FUNCTION_BLOCK FB_ROB_AMR EXTENDS FB_ROB IMPLEMENTS ITF_2_AMR
VAR_INPUT
END_VAR
VAR_OUTPUT
	visStatus: stVisStatusAMR;
	bTargetreached: BOOL;
END_VAR
VAR
	_tcppos, _tcpvel : stPose2D;
	_jointpos, _jointvel: stJoint2;
	
END_VAR

{warning 'Add property implementation'}
PROPERTY ActualJointPosition : stJoint2
GET
ActualJointPosition := _jointpos;
END_GET
END_PROPERTY

{warning 'Add property implementation'}
PROPERTY ActualJointVelocity : stJoint2
GET
ActualJointVelocity:= _jointvel;
END_GET
END_PROPERTY

{warning 'Add property implementation'}
PROPERTY ActualTcpPose : stPose2D
GET
ActualTcpPose := _tcppos;
END_GET
END_PROPERTY

{warning 'Add property implementation'}
PROPERTY ActualTcpVelocity : stPose2D
GET
ActualTcpVelocity := _tcpvel;
END_GET
END_PROPERTY

ACTION CYCLIC_AMR:
CYCLIC_ROB();

visStatus.State:=eStatus;
visStatus.Mode:=eModus;
visStatus.isMoving:=RobotMoving;
visStatus.isReady:=RobotReady;
visStatus.isConnected:=CommunicationReady;
// 	isLocked: BOOL;
// visStatus.isBusy:=;
visStatus.isInCollision:=Collision;
visStatus.hasError:=bError;
visStatus.TCPPosition:=ActualTcpPose;

visStatus.isDocked:=IsDocked;
visStatus.TargetReached:=TargetReached;
END_ACTION

METHOD Dock : BOOL
END_METHOD

{warning 'Add property implementation'}
PROPERTY IsDocked : BOOL
GET
END_GET
END_PROPERTY

// {warning 'Add method implementation '}
  METHOD NavigateToGoal : BOOL
VAR_INPUT
    goal : STRING;
END_VAR
END_METHOD

METHOD NavigateToPoint : BOOL
  VAR_INPUT
    point : stPose2D;
  END_VAR
END_METHOD

METHOD PROTECTED OnActivate : eResult
IF bError THEN
    OnActivate := eResult.ERROR;
    ELSIF CommunicationReady THEN
      OnActivate := eResult.SUCCESS;
ELSE
      OnActivate := eResult.None;
END_IF
END_METHOD

METHOD PROTECTED OnCleanup : eResult
// Disconnect();
// 
//     IF eConnectionState <> eCommunicationState.DISCONNECTED THEN
//       OnCleanup := eResult.None;
//     ELSE
      OnCleanup := eResult.SUCCESS;
//     END_IF
END_METHOD

METHOD PROTECTED OnConfigure : eResult

PM.Configure(sPrefix:=Name,sDatabase:=CONCAT('db_',Name));

// if fbPM.b

OnConfigure := eResult.SUCCESS;
END_METHOD

METHOD PROTECTED OnDeactivate : eResult
IF bError THEN
    OnDeactivate := eResult.ERROR;
ELSE
    OnDeactivate := eResult.SUCCESS;
END_IF
END_METHOD

METHOD PROTECTED OnError : eResult
OnError := eResult.SUCCESS;
END_METHOD

METHOD PROTECTED OnShutdown : eResult
// Disconnect();
// 
//     IF eConnectionState <> eCommunicationState.DISCONNECTED THEN
//       OnShutdown := eResult.None;
//     ELSIF bError THEN
//       OnShutdown := eResult.ERROR;
//     ELSE
      OnShutdown := eResult.SUCCESS;
//     END_IF
END_METHOD

PROPERTY TargetReached : BOOL
GET
TargetReached:=bTargetreached;
END_GET
SET
bTargetreached:=TargetReached;
END_SET
END_PROPERTY

METHOD Undock : BOOL
  VAR_INPUT
  END_VAR
END_METHOD

END_FUNCTION_BLOCK

(* stored: Version 1.1.0.1, ProductVersion 3.1.4026.18
   POU FB_ROB_AMR: Id {cf71feff-3eb8-4d62-9de2-ec89e7c3ba43}, SpecialFunc None
   Folder MotionControl - Override: Id {67b3627f-d3d9-4d23-986a-0e1d03e05b51}
   Folder StateControl: Id {5824b502-00ae-4537-9581-ce8706661f80}
   Property ActualJointPosition: Id {a9bb0008-2bc7-471b-b7cd-69232649304e}
   Get Get: Id {c40e1322-8cf0-4659-99cb-1ad8b6629bcb}
   Property ActualJointVelocity: Id {0493ea03-284e-4697-b6d9-85f06afe56ed}
   Get Get: Id {6f83ad7c-bb1b-49e3-a3b5-2da802613af4}
   Property ActualTcpPose: Id {5f2eea29-65d5-4ce1-8b21-86b7c8473be6}
   Get Get: Id {fa0df135-1f19-4fd2-b0d5-1f3480c883d6}
   Property ActualTcpVelocity: Id {353dfdcb-eeca-4ed7-9a9e-990541ee5c2e}
   Get Get: Id {edff15a4-fbcc-4630-ae2a-c4883c3e01f6}
   Action CYCLIC_AMR: Id {ebcfe1a2-a428-4cd0-a9d1-512be0cd10b6}
   Method Dock: Id {7a2cbcfa-840f-4b61-9db6-42db4be3c502}
   Property IsDocked: Id {b1223d7e-f467-499a-a850-c3753fbde900}
   Get Get: Id {4fc975e3-63b2-4f01-8d05-8125246e628b}
   Method NavigateToGoal: Id {b2e2ff45-ccbe-41b1-afea-be4075ff97b2}
   Method NavigateToPoint: Id {2db64f24-9a85-44a5-a853-3b922490bedd}
   Method OnActivate: Id {87bcfeb5-637b-4246-b013-c7747d0d3053}
   Method OnCleanup: Id {70dc0820-01d4-4f5b-84fc-9914b0c296bf}
   Method OnConfigure: Id {cb165446-431a-4f44-a815-7e6356f9994b}
   Method OnDeactivate: Id {53f91d36-ca4e-4655-9369-60aadeb29812}
   Method OnError: Id {d2189026-696b-4a07-b8cf-376dec470a43}
   Method OnShutdown: Id {04379ee7-470c-4f20-91e9-ed3450a5b8b5}
   Property TargetReached: Id {1ffd5e85-127b-44be-a405-ac0615b395e0}
   Get Get: Id {57de425a-d48b-4d0b-8603-0f3a7e17fce2}
   Set Set: Id {942b15fc-f5de-4bca-9fdf-4d667e329064}
   Method Undock: Id {7fd604b3-b44b-4e9a-9b9f-e9b2cbe8020e} *)
